DATA_BLOCK "11_PB_Released"
{ DB_Accessible_From_OPC_UA := 'FALSE' ;
 S7_Optimized_Access := 'TRUE' }
VERSION : 0.1
NON_RETAIN
   VAR
      "S1+MS1+ES2028-SF3222_PB" { ExternalWritable := 'False'} : Bool;
   END_VAR


BEGIN

END_DATA_BLOCK

